TYPE DS_EventHistory EXTENDS DS_Event :
STRUCT
	sTimeAndDate_Recovered 			: STRING(50);
	sTimeAndDate_Acknowledged 		: STRING(50);
	
END_STRUCT
END_TYPE

(* stored: Version 1.1.0.1, ProductVersion 3.1.4024.12
   DUT DS_EventHistory: Id {cc348f9e-f74e-4643-a07c-0cbe18c2f575} *)
